TYPE DUT_stUpdateBatchToProductionQueue :
STRUCT
	return_			: DINT;
	BatchId	: STRING(DB.MAX_STRING_SIZE);
	BatchInfoJson	: STRING(DB.MAX_STRING_SIZE);
	BatchItemsJson	: STRING(DB.MAX_STRING_SIZE);
END_STRUCT
END_TYPE

(* stored: Version 1.1.0.1, ProductVersion 3.1.4024.15
   DUT DUT_stUpdateBatchToProductionQueue: Id {14b58b27-634e-4166-927d-9086aca60a02} *)
